// TIA Portal project "FactoryIOElevatorAdvanced" (V15.1)

(* hardware
DEVICE "S7-1200 station_1"  S7-1200 Station
   slot 0: "Rack_0"  S7-1200 Rack  Rack  V1.0
   slot 1: "PLC_1"  CPU 1212C DC/DC/DC  6ES7 212-1AE40-0XB0  V4.2
*)

// ===== PLC "PLC_1"  CPU 1212C DC/DC/DC =====

VAR_GLOBAL   // PLC tag table "Default tag table"
   "START" AT %I1.6 : Bool;
   "Esteira 0" AT %Q0.0 : Bool;
   "LIGADO" AT %M0.0 : Bool;
   "STOP" AT %I2.0 : Bool;
   "Sen. Sobre Elev." AT %I2.5 : Bool;
   "Esteira 1" AT %Q0.1 : Bool;
   "Sen. Entrada Elev." AT %I2.4 : Bool;
   "Carregando" AT %M0.1 : Bool;
   "Up" AT %Q0.7 : Bool;
   "N0 (low)" AT %I0.6 : Bool;
   "N0 (high)" AT %I0.7 : Bool;
   "N1 (low)" AT %I1.0 : Bool;
   "N1 (high)" AT %I1.1 : Bool;
   "N2 (low)" AT %I1.2 : Bool;
   "N2 (high)" AT %I1.3 : Bool;
   "N3 (low)" AT %I1.4 : Bool;
   "N3 (high)" AT %I1.5 : Bool;
   "Slow" AT %Q1.1 : Bool;
   "Esteira 2" AT %Q0.2 : Bool;
   "Esteira 3" AT %Q0.3 : Bool;
   "Sen. Placa 1" AT %I2.7 : Bool;
   "Sen. Placa 2" AT %I3.0 : Bool;
   "Sen. Placa 3" AT %I3.1 : Bool;
   "Emergency" AT %I2.1 : Bool;
   "Reset" AT %I1.7 : Bool;
   "Carregado" AT %M0.2 : Bool;
   "Esteira Flag" AT %M0.3 : Bool;
   "Placa descendo" AT %M0.4 : Bool;
   "Próximo passo" AT %M0.5 : Bool;
   "Tag_1" AT %M0.6 : Bool;
   "Finalizou" AT %M0.7 : Bool;
   "Down" AT %Q1.0 : Bool;
   "Esteira Elev." AT %Q0.5 : Bool;
   "Sen. Saída Elev." AT %I2.6 : Bool;
END_VAR

DATA_BLOCK "DB"   // DB1
{ S7_Optimized_Access := 'TRUE' }
VERSION : 0.1
   VAR
      "M" : Array[0..17] of Bool;
      Ligado : Bool;
   END_VAR
BEGIN
END_DATA_BLOCK

// folder: System blocks/Program resources

DATA_BLOCK "Time 1"   // DB2
{ S7_Optimized_Access := 'TRUE' }
AUTHOR : Simatic
FAMILY : IEC
NAME : IEC_TMR
VERSION : 1.0
// stored: InstanceOfName IEC_TIMER
"IEC_TIMER"
BEGIN
END_DATA_BLOCK

DATA_BLOCK "Timer 2"   // DB3
{ S7_Optimized_Access := 'TRUE' }
AUTHOR : Simatic
FAMILY : IEC
NAME : IEC_TMR
VERSION : 1.0
// stored: InstanceOfName IEC_TIMER
"IEC_TIMER"
BEGIN
END_DATA_BLOCK

DATA_BLOCK "Timer 4"   // DB4
{ S7_Optimized_Access := 'TRUE' }
AUTHOR : Simatic
FAMILY : IEC
NAME : IEC_TMR
VERSION : 1.0
// stored: InstanceOfName IEC_TIMER
"IEC_TIMER"
BEGIN
END_DATA_BLOCK

DATA_BLOCK "Timer 3"   // DB5
{ S7_Optimized_Access := 'TRUE' }
AUTHOR : Simatic
FAMILY : IEC
NAME : IEC_TMR
VERSION : 1.0
// stored: InstanceOfName IEC_TIMER
"IEC_TIMER"
BEGIN
END_DATA_BLOCK

DATA_BLOCK "Timer 5"   // DB6
{ S7_Optimized_Access := 'TRUE' }
AUTHOR : Simatic
FAMILY : IEC
NAME : IEC_TMR
VERSION : 1.0
// stored: InstanceOfName IEC_TIMER
"IEC_TIMER"
BEGIN
END_DATA_BLOCK

DATA_BLOCK "Timer 6"   // DB7
{ S7_Optimized_Access := 'TRUE' }
AUTHOR : Simatic
FAMILY : IEC
NAME : IEC_TMR
VERSION : 1.0
// stored: InstanceOfName IEC_TIMER
"IEC_TIMER"
BEGIN
END_DATA_BLOCK

DATA_BLOCK "Timer 7"   // DB8
{ S7_Optimized_Access := 'TRUE' }
AUTHOR : Simatic
FAMILY : IEC
NAME : IEC_TMR
VERSION : 1.0
// stored: InstanceOfName IEC_TIMER
"IEC_TIMER"
BEGIN
END_DATA_BLOCK

// folder: (top level)

FUNCTION "MHJ-PLC-Lab-Function-S71200" : Void   // FC9000, SCL
{ S7_Optimized_Access := 'TRUE' }
VERSION : 0.1
   VAR_TEMP
      rdTimeReturn : Int;
      outputTime : DTL;
      SyncVal : Byte;
      forVal : Int;
      forVal_2 : Int;
      Value : Byte;
   END_VAR
   VAR CONSTANT
      CompVal : Byte := 16#34;
      Value_01 : Byte := 16#11;
      Value_01_DW : DWord := 16#A165_D992;
      Value_02_DW : DWord := 16#58BE_4401;
   END_VAR
BEGIN

   #Value:=PEEK(area := 16#82,
        dbNumber := 0,
        byteOffset := 511);
   #Value := #Value + 1;

   POKE(area := 16#82,
        dbNumber := 0,
        byteOffset := 511,
        value := #Value);

   POKE(area:=16#81,
        dbNumber:=0,
        byteOffset:=1016,
        value:=#Value_01_DW);
   POKE(area := 16#81,
        dbNumber := 0,
        byteOffset := 1020,
        value := #Value_02_DW);

   POKE(area := 16#81,
        dbNumber := 0,
        byteOffset := 511,
        value := B#16#00);

   FOR #forVal := 0 TO 120 DO
       FOR #forVal_2:=0 TO 10 DO
           #rdTimeReturn:=RD_SYS_T(#outputTime);
           #rdTimeReturn := WR_SYS_T(#outputTime);
           #rdTimeReturn := RD_SYS_T(#outputTime);
           #rdTimeReturn := WR_SYS_T(#outputTime);
       END_FOR;
       #SyncVal:= PEEK(area := 16#81,
                      dbNumber := 0,
                      byteOffset := 511);
       IF #SyncVal = #CompVal THEN
          GOTO M_1;
       END_IF;
   END_FOR;
   RETURN;

   M_1:
   POKE(area := 16#81,
        dbNumber := 0,
        byteOffset := 511,
        value := B#16#0);
END_FUNCTION

ORGANIZATION_BLOCK "Main"   // OB1, LAD, ProgramCycle
TITLE = "Main Program Sweep (Cycle)"
{ S7_Optimized_Access := 'TRUE' }
VERSION : 0.1
   VAR_INPUT
      Initial_Call : Bool;   // Initial call of this OB
      Remanence : Bool;   // =True, if remanent data are available
   END_VAR
   VAR_TEMP   // added for the SCL form of the ladder/FBD networks
      _w1 : Bool;
      _w2 : Bool;
   END_VAR
BEGIN

REGION Network 1
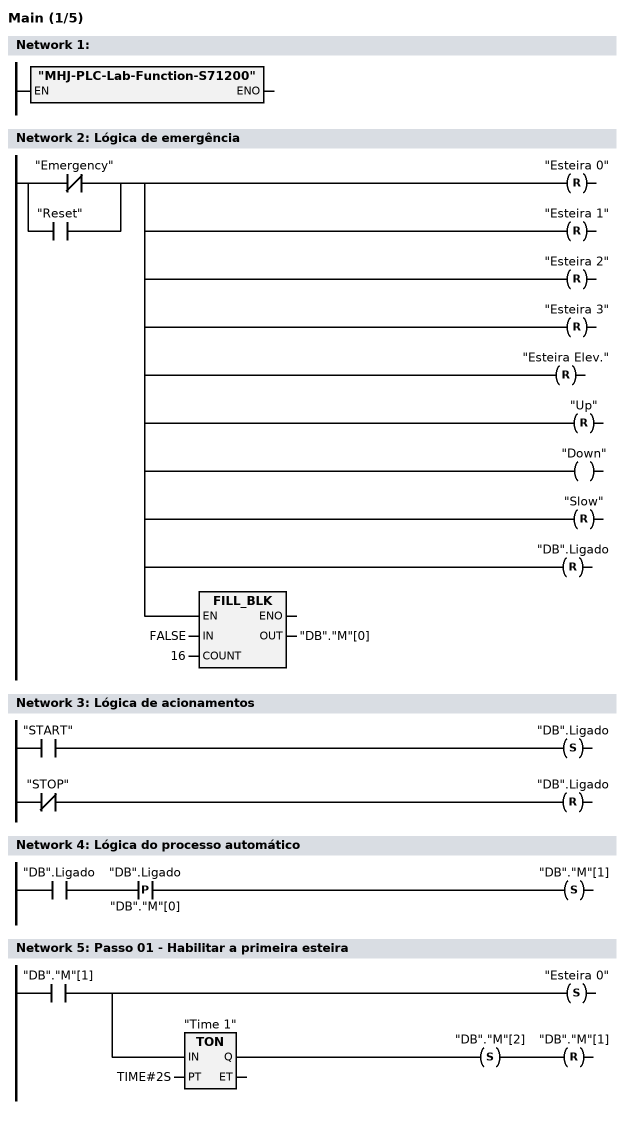
   RUNG wire#powerrail
      "MHJ-PLC-Lab-Function-S71200"()
   END_RUNG
   // the same network as SCL:
   "MHJ-PLC-Lab-Function-S71200"();
END_REGION

REGION Network 2: Lógica de emergência
   RUNG wire#powerrail
      I_Contact( "Emergency" )
      wire#w1
      R_Coil( "Esteira 0" )
   END_RUNG
   RUNG wire#powerrail
      Contact( "Reset" )
   END_RUNG wire#w1
   RUNG wire#w1
      R_Coil( "Esteira 1" )
   END_RUNG
   RUNG wire#w1
      R_Coil( "Esteira 2" )
   END_RUNG
   RUNG wire#w1
      R_Coil( "Esteira 3" )
   END_RUNG
   RUNG wire#w1
      R_Coil( "Esteira Elev." )
   END_RUNG
   RUNG wire#w1
      R_Coil( "Up" )
   END_RUNG
   RUNG wire#w1
      Coil( "Down" )
   END_RUNG
   RUNG wire#w1
      R_Coil( "Slow" )
   END_RUNG
   RUNG wire#w1
      R_Coil( "DB".Ligado )
   END_RUNG
   RUNG wire#w1
      FillBlockI(in := FALSE, count := 16, out => "DB"."M"[0])
   END_RUNG
   // the same network as SCL:
   #_w1 := NOT "Emergency" OR "Reset";
   IF #_w1 THEN
       "Esteira 0" := FALSE;
       "Esteira 1" := FALSE;
       "Esteira 2" := FALSE;
       "Esteira 3" := FALSE;
       "Esteira Elev." := FALSE;
       "Up" := FALSE;
   END_IF;
   "Down" := #_w1;
   IF #_w1 THEN
       "Slow" := FALSE;
       "DB".Ligado := FALSE;
       FILL_BLK(IN := FALSE, COUNT := 16, OUT => "DB"."M"[0]);
   END_IF;
END_REGION

REGION Network 3: Lógica de acionamentos
   RUNG wire#powerrail
      Contact( "START" )
      S_Coil( "DB".Ligado )
   END_RUNG
   RUNG wire#powerrail
      I_Contact( "STOP" )
      R_Coil( "DB".Ligado )
   END_RUNG
   // the same network as SCL:
   IF "START" THEN "DB".Ligado := TRUE; END_IF;
   IF NOT "STOP" THEN "DB".Ligado := FALSE; END_IF;
END_REGION

REGION Network 4: Lógica do processo automático
   RUNG wire#powerrail
      Contact( "DB".Ligado )
      P_Contact(operand := "DB".Ligado, bit := "DB"."M"[0])
      S_Coil( "DB"."M"[1] )
   END_RUNG
   // the same network as SCL:
   #_w1 := "DB".Ligado AND "DB".Ligado AND NOT "DB"."M"[0];   // rising edge of "DB".Ligado
   "DB"."M"[0] := "DB".Ligado;
   IF #_w1 THEN "DB"."M"[1] := TRUE; END_IF;
END_REGION

REGION Network 5: Passo 01 - Habilitar a primeira esteira
   IF "DB"."M"[1] THEN "Esteira 0" := TRUE; END_IF;
   "Time 1".TON(IN := "DB"."M"[1], PT := TIME#2S);
   IF "Time 1".Q THEN
       "DB"."M"[2] := TRUE;
       "DB"."M"[1] := FALSE;
   END_IF;
END_REGION

REGION Network 6: Passo 02 - Caixa carregada no elevador
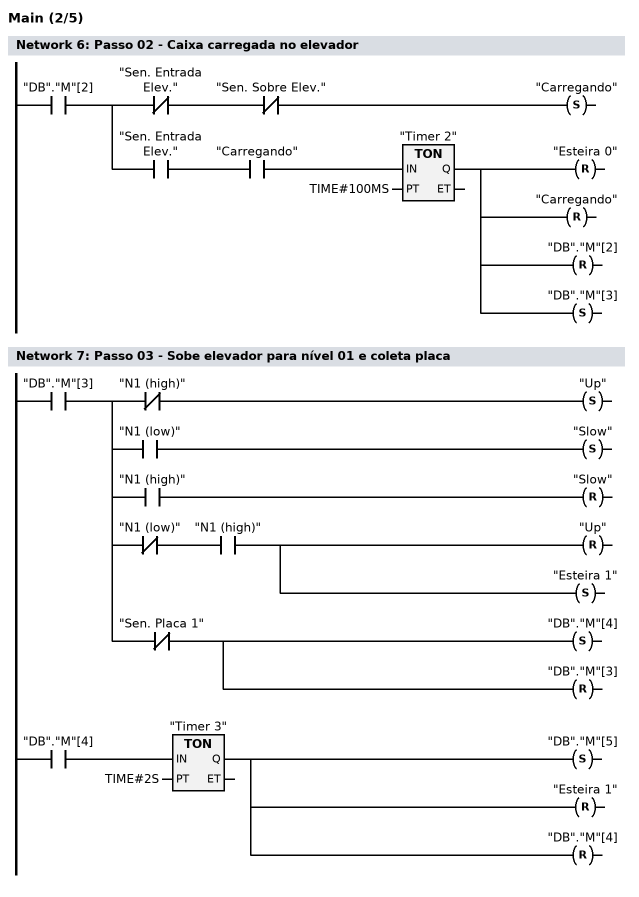
   IF "DB"."M"[2] AND NOT "Sen. Entrada Elev." AND NOT "Sen. Sobre Elev." THEN "Carregando" := TRUE; END_IF;
   "Timer 2".TON(IN := "DB"."M"[2] AND "Sen. Entrada Elev." AND "Carregando", PT := TIME#100MS);
   IF "Timer 2".Q THEN
       "Esteira 0" := FALSE;
       "Carregando" := FALSE;
       "DB"."M"[2] := FALSE;
       "DB"."M"[3] := TRUE;
   END_IF;
END_REGION

REGION Network 7: Passo 03 - Sobe elevador para nível 01 e coleta placa
   IF "DB"."M"[3] AND NOT "N1 (high)" THEN "Up" := TRUE; END_IF;
   IF "DB"."M"[3] AND "N1 (low)" THEN "Slow" := TRUE; END_IF;
   IF "DB"."M"[3] AND "N1 (high)" THEN "Slow" := FALSE; END_IF;
   IF "DB"."M"[3] AND NOT "N1 (low)" AND "N1 (high)" THEN
       "Up" := FALSE;
       "Esteira 1" := TRUE;
   END_IF;
   #_w1 := "DB"."M"[3] AND NOT "Sen. Placa 1";
   IF #_w1 THEN
       "DB"."M"[4] := TRUE;
       "DB"."M"[3] := FALSE;
   END_IF;
   "Timer 3".TON(IN := "DB"."M"[4], PT := TIME#2S);
   IF "Timer 3".Q THEN
       "DB"."M"[5] := TRUE;
       "Esteira 1" := FALSE;
       "DB"."M"[4] := FALSE;
   END_IF;
END_REGION

REGION Network 8: Passo 04 - Sobe elevador para nível 02 e coleta placa
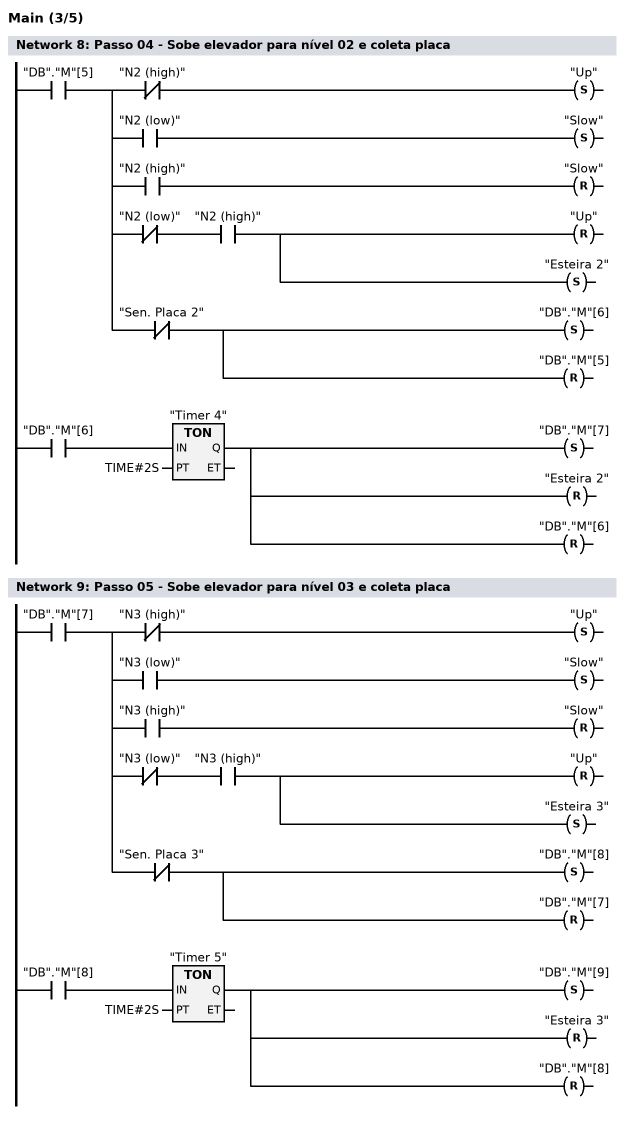
   IF "DB"."M"[5] AND NOT "N2 (high)" THEN "Up" := TRUE; END_IF;
   IF "DB"."M"[5] AND "N2 (low)" THEN "Slow" := TRUE; END_IF;
   IF "DB"."M"[5] AND "N2 (high)" THEN "Slow" := FALSE; END_IF;
   IF "DB"."M"[5] AND NOT "N2 (low)" AND "N2 (high)" THEN
       "Up" := FALSE;
       "Esteira 2" := TRUE;
   END_IF;
   #_w1 := "DB"."M"[5] AND NOT "Sen. Placa 2";
   IF #_w1 THEN
       "DB"."M"[6] := TRUE;
       "DB"."M"[5] := FALSE;
   END_IF;
   "Timer 4".TON(IN := "DB"."M"[6], PT := TIME#2S);
   IF "Timer 4".Q THEN
       "DB"."M"[7] := TRUE;
       "Esteira 2" := FALSE;
       "DB"."M"[6] := FALSE;
   END_IF;
END_REGION

REGION Network 9: Passo 05 - Sobe elevador para nível 03 e coleta placa
   IF "DB"."M"[7] AND NOT "N3 (high)" THEN "Up" := TRUE; END_IF;
   IF "DB"."M"[7] AND "N3 (low)" THEN "Slow" := TRUE; END_IF;
   IF "DB"."M"[7] AND "N3 (high)" THEN "Slow" := FALSE; END_IF;
   IF "DB"."M"[7] AND NOT "N3 (low)" AND "N3 (high)" THEN
       "Up" := FALSE;
       "Esteira 3" := TRUE;
   END_IF;
   #_w1 := "DB"."M"[7] AND NOT "Sen. Placa 3";
   IF #_w1 THEN
       "DB"."M"[8] := TRUE;
       "DB"."M"[7] := FALSE;
   END_IF;
   "Timer 5".TON(IN := "DB"."M"[8], PT := TIME#2S);
   IF "Timer 5".Q THEN
       "DB"."M"[9] := TRUE;
       "Esteira 3" := FALSE;
       "DB"."M"[8] := FALSE;
   END_IF;
END_REGION

REGION Network 10: Passo 06 - Desce elevador para nível 02 e coleta placa
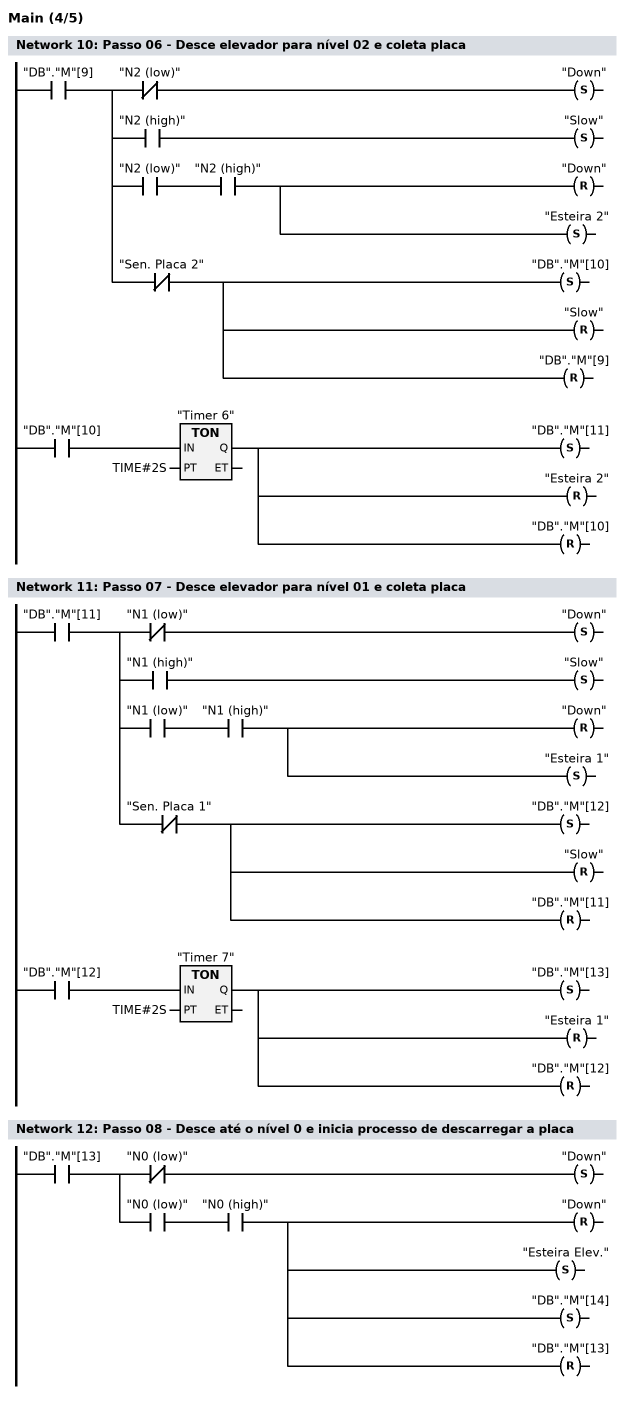
   IF "DB"."M"[9] AND NOT "N2 (low)" THEN "Down" := TRUE; END_IF;
   IF "DB"."M"[9] AND "N2 (high)" THEN "Slow" := TRUE; END_IF;
   IF "DB"."M"[9] AND "N2 (low)" AND "N2 (high)" THEN
       "Down" := FALSE;
       "Esteira 2" := TRUE;
   END_IF;
   #_w1 := "DB"."M"[9] AND NOT "Sen. Placa 2";
   IF #_w1 THEN
       "DB"."M"[10] := TRUE;
       "Slow" := FALSE;
       "DB"."M"[9] := FALSE;
   END_IF;
   "Timer 6".TON(IN := "DB"."M"[10], PT := TIME#2S);
   IF "Timer 6".Q THEN
       "DB"."M"[11] := TRUE;
       "Esteira 2" := FALSE;
       "DB"."M"[10] := FALSE;
   END_IF;
END_REGION

REGION Network 11: Passo 07 - Desce elevador para nível 01 e coleta placa
   IF "DB"."M"[11] AND NOT "N1 (low)" THEN "Down" := TRUE; END_IF;
   IF "DB"."M"[11] AND "N1 (high)" THEN "Slow" := TRUE; END_IF;
   IF "DB"."M"[11] AND "N1 (low)" AND "N1 (high)" THEN
       "Down" := FALSE;
       "Esteira 1" := TRUE;
   END_IF;
   #_w1 := "DB"."M"[11] AND NOT "Sen. Placa 1";
   IF #_w1 THEN
       "DB"."M"[12] := TRUE;
       "Slow" := FALSE;
       "DB"."M"[11] := FALSE;
   END_IF;
   "Timer 7".TON(IN := "DB"."M"[12], PT := TIME#2S);
   IF "Timer 7".Q THEN
       "DB"."M"[13] := TRUE;
       "Esteira 1" := FALSE;
       "DB"."M"[12] := FALSE;
   END_IF;
END_REGION

REGION Network 12: Passo 08 - Desce até o nível 0 e inicia processo de descarregar a placa
   RUNG wire#powerrail
      Contact( "DB"."M"[13] )
      wire#w1
      I_Contact( "N0 (low)" )
      S_Coil( "Down" )
   END_RUNG
   RUNG wire#w1
      Contact( "N0 (low)" )
      Contact( "N0 (high)" )
      wire#w2
      R_Coil( "Down" )
   END_RUNG
   RUNG wire#w2
      S_Coil( "Esteira Elev." )
   END_RUNG
   RUNG wire#w2
      S_Coil( "DB"."M"[14] )
   END_RUNG
   RUNG wire#w2
      R_Coil( "DB"."M"[13] )
   END_RUNG
   // the same network as SCL:
   IF "DB"."M"[13] AND NOT "N0 (low)" THEN "Down" := TRUE; END_IF;
   IF "DB"."M"[13] AND "N0 (low)" AND "N0 (high)" THEN
       "Down" := FALSE;
       "Esteira Elev." := TRUE;
   END_IF;
   #_w1 := "DB"."M"[13] AND "N0 (low)" AND "N0 (high)";
   IF #_w1 THEN
       "DB"."M"[14] := TRUE;
       "DB"."M"[13] := FALSE;
   END_IF;
END_REGION

REGION Network 13: Passo 09 - Verifica se a caixa foi descarregada e reinicia
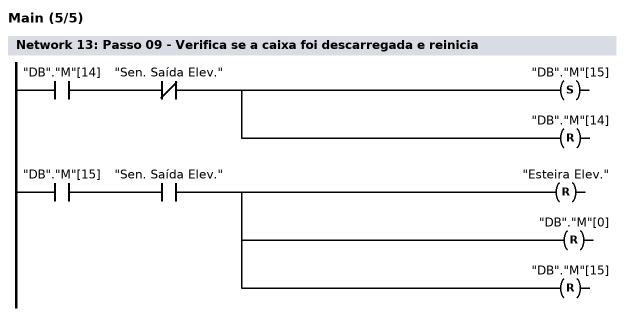
   RUNG wire#powerrail
      Contact( "DB"."M"[14] )
      I_Contact( "Sen. Saída Elev." )
      wire#w1
      S_Coil( "DB"."M"[15] )
   END_RUNG
   RUNG wire#w1
      R_Coil( "DB"."M"[14] )
   END_RUNG
   RUNG wire#powerrail
      Contact( "DB"."M"[15] )
      Contact( "Sen. Saída Elev." )
      wire#w2
      R_Coil( "Esteira Elev." )
   END_RUNG
   RUNG wire#w2
      R_Coil( "DB"."M"[0] )
   END_RUNG
   RUNG wire#w2
      R_Coil( "DB"."M"[15] )
   END_RUNG
   // the same network as SCL:
   #_w1 := "DB"."M"[14] AND NOT "Sen. Saída Elev.";
   IF #_w1 THEN
       "DB"."M"[15] := TRUE;
       "DB"."M"[14] := FALSE;
   END_IF;
   IF "DB"."M"[15] AND "Sen. Saída Elev." THEN "Esteira Elev." := FALSE; END_IF;
   #_w2 := "DB"."M"[15] AND "Sen. Saída Elev.";
   IF #_w2 THEN
       "DB"."M"[0] := FALSE;
       "DB"."M"[15] := FALSE;
   END_IF;
END_REGION
END_ORGANIZATION_BLOCK